FUNCTION "bioTransMan" : Void
TITLE = Batch I/O Transfer Manager
{ S7_Optimized_Access := 'TRUE' }
AUTHOR : Woermann
VERSION : 0.1
// -- Woermann Automation --
//Block to Unify and Manage Transfer Communication Signals
	VAR_INPUT
		Master : Bool;   // True if this is the Transfer Master
		LocalID : DInt;   // Local ID like PrID or selected Equipment
		PartnerID : DInt;   // Partner ID like PrID or Equipment
	END_VAR

	VAR_OUTPUT
		Start : Bool;   // Start Transfer
	END_VAR

	VAR_IN_OUT
		rtRec : Bool;   // Ready to Receive
		rtSnd : Bool;   // Ready to Send
		reRec : Bool;   // Release / Request Receive
		reSnd : Bool;   // Release / Request Send
	END_VAR


BEGIN
NETWORK
TITLE =
END_FUNCTION

